Staubli VAL3: getVariance.pgx

public program getVariance(num& x_nInput[], num& x_nVariance)
  local num l_nMean
  local num l_nCount
  local num l_nSum
begin

  l_nSum = 0
  // get mean of the input numbers
  call getMean(x_nInput, l_nMean)

  for l_nCount = 0 to size(x_nInput)-1
    l_nSum = l_nSum + power(x_nInput[l_nCount]-l_nMean, 2)
  endFor

  x_nVariance = l_nSum/size(x_nInput)

end
